TYPE POSITION :
STRUCT
	X : LREAL;
	Y : LREAL;
	Z : LREAL;
END_STRUCT
END_TYPE

(* stored: Version 1.1.0.1, ProductVersion 3.1.4020.3
   DUT POSITION: Id {dd308c4c-e62f-48d3-984d-9cfc2c186943} *)
